screen "S2 Manual Mode" 1280x700, template "Navigation"
   on ClearScreen: SetBit("S2 Setup Data_Leave Manual Screen")
   on GenerateScreen: ResetBit("S2 Setup Data_Leave Manual Screen")
   Group "Group_3" at 492,12 size 427x42; Text 'SYSTEM 1'
   Group "Group_10" at 1149,100 size 112x111; Authorization "Health_Physics"
   Switch "Pushbutton_Emergency_1" at 935,29 size 60x61; CaptionText 'Switch'; TextOff '0'; TextOn '1'; PictureOff "Pushbutton_Emergency_Off_256c"; PictureOn "Pushbutton_Emergency_On_256c"
      Visibility <- "Station 2 Estop PB Active"
      ProcessValue <- "Station 2 Estop PB Active"
   TextField "Text field_53" at 933,7 size 65x25; Text 'ESTOP'
      Visibility <- "Station 2 Estop PB Active"
   Rectangle "Rectangle_4" at 411,100 size 720x467
      Appearance <- "Station 2 Run State"
   SymbolLibrary "Symbol library_18" at 680,195 size 148x16
      Appearance <- "Station 2 Tubing Rinse"
   SymbolLibrary "Symbol library_13" at 840,222 size 15x255
      Appearance <- "Station 2 Pump Tubing"
   SymbolLibrary "Symbol library_2" at 553,234 size 298x124
   SymbolLibrary "Symbol library_21" at 869,195 size 116x16
      Appearance <- "Station 2 Tubing Drain"
   TextField "Text field_9" at 590,186 size 85x32; Text 'RINSE'
   TextField "Text field_10" at 983,170 size 151x32; Text 'UNWANTED'
   TextField "Text field_14" at 828,471 size 38x32; Text 'SV'
   Group "Group_6" at 816,158 size 65x82
   Group "Group_12" at 916,230 size 108x188; TextOff 'WASTE'
   Group "Group_11" at 995,442 size 114x111; Authorization "Maintenance"
   TextField "Text field_17" at 984,192 size 135x32; Text 'MATERIAL'
   Group "Group" at 436,425 size 144x122
   Group "Group_4" at 629,370 size 156x40
   Group "Group_13" at 596,422 size 219x134; Text 'PUMP SPEED'; FormatPattern 99999
   Group "Group_14" at 1151,219 size 120x111; TextOff 'BYPASS'; Text 'DOOR LOCK'
   Group "Group_15" at 436,227 size 105x188
   Group "Group_9" at 482,274 size 532x42; Text 'SYSTEM 1'
   Group "Group_17" at 185,13 size 215x125; Authorization "Maintenance"
   IOField "I/O field_2" at 629,96 size 159x56; FormatPattern 9999.9
      ProcessValue <- "Station 2 MM Feedback RPM"
   TextField "Text field_8" at 629,64 size 165x32; Text 'PUMP SPEED'
   Rectangle "Rectangle_16" at 631,99 size 154x49
      Visibility <- "Station 2 Manual Mode"
   TextField "Text field_11" at 672,150 size 61x32; Text 'RPM'
   Group "Group_16" at 615,272 size 194x44
   Group "Group_18" at 615,272 size 194x44
   Group "Group_19" at 561,579 size 419x93
   Group "Group_20" at 561,579 size 419x93
   TextField "Text field_13" at 502,12 size 417x39; Text 'STATION 2 MANUAL MODE'
   Rectangle "Rectangle_11" at 482,274 size 518x42
      Visibility <- "Station 2 Process Running"
   TextField "Text field_16" at 494,274 size 520x39; Text 'STATION 2 IN AUTOMATIC MODE'
      Visibility <- "Station 2 Process Running"
   Rectangle "Rectangle_13" at 1149,100 size 112x111
      Visibility <- "CurrentGroupNum"
   TextField "Text field_15" at 1158,104 size 97x23; Text 'RAD LOCK'
      Visibility <- "CurrentGroupNum"
   Button "Button_15" at 1164,130 size 80x70; TextOff 'BYPASS'; Authorization "Health_Physics"
      on Press: InvertBit("Station 2 Rad Lock Bypass")
      Visibility <- "CurrentGroupNum"
   GraphicIOField "PlotLight_Round_GN_6" at 1218,132 size 22x23; PictureOn "PilotLight_Round_GN_On_256c"; PictureOff "PilotLight_Round_GN_Off_256c"; Authorization "Health_Physics"
      Visibility <- "CurrentGroupNum"
      ProcessValue <- "Station 2 Rad Lock Bypass"
   Group "Group_1" at 596,422 size 219x134; Text 'PUMP SPEED'; FormatPattern 99999
   Rectangle "Rectangle_12" at 629,463 size 154x49
      Visibility <- "Station 2 Manual Mode"
   IOField "I/O field_1" at 626,460 size 159x56; FormatPattern 9999.9
      ProcessValue <- "Station 2 Pump Speed RPM SP"
   TextField "Text field_5" at 607,428 size 205x32; Text 'PUMP SPEED SP'
   TextField "Text field_7" at 670,518 size 61x32; Text 'RPM'
   SymbolLibrary "Symbol library_4" at 816,185 size 32x36
      Appearance <- "Station 2 Valve Rinse"
   SymbolLibrary "Symbol library_3" at 849,185 size 32x36
      Appearance <- "Station 2 Valve Drain"
   SymbolLibrary "Symbol library_5" at 832,204 size 32x36
      Appearance <- "Station 2 Valve Pump"
   Group "Group_5" at 436,227 size 105x188
   Button "Button_9" at 449,264 size 74x63; TextOff 'FWD'
      Visibility <- "Station 2 Manual Mode"
   Button "Button_10" at 451,343 size 74x63; TextOff 'REV'
      Visibility <- "Station 2 Manual Mode"
   TextField "Text field_3" at 448,230 size 77x32; Text 'PUMP'
   Button "Button_5" at 449,264 size 74x63; TextOff 'FWD'
      on Press: SetBit("Station 2 MM Pump Dir FWD"); ResetBit("Station 2 MM Pump Dir REV")
   Button "Button_6" at 451,343 size 74x63; TextOff 'REV'
      on Press: SetBit("Station 2 MM Pump Dir REV"); ResetBit("Station 2 MM Pump Dir FWD")
   GraphicIOField "PlotLight_Round_GN_2" at 501,345 size 22x23; PictureOn "PilotLight_Round_GN_On_256c"; PictureOff "PilotLight_Round_GN_Off_256c"
      ProcessValue <- "Station 2 MM Pump Dir REV"
   GraphicIOField "PlotLight_Round_GN_5" at 500,266 size 22x23; PictureOn "PilotLight_Round_GN_On_256c"; PictureOff "PilotLight_Round_GN_Off_256c"
      ProcessValue <- "Station 2 MM Pump Dir FWD"
   Group "Group_2" at 916,230 size 108x188; TextOff 'WASTE'
   Button "Button_11" at 930,267 size 74x63; TextOff 'UM'
      Visibility <- "Station 2 Manual Mode"
   Button "Button_12" at 930,345 size 74x63; TextOff 'RINSE'
      Visibility <- "Station 2 Manual Mode"
   TextField "Text field_6" at 924,232 size 85x32; Text 'VALVE'
   Button "Button_7" at 930,267 size 74x63; TextOff 'UM'
      on Press: ResetBit("Station 2 MM Valve Direction SW")
   Button "Button_8" at 930,345 size 74x63; TextOff 'RINSE'
      on Press: SetBit("Station 2 MM Valve Direction SW")
   GraphicIOField "PlotLight_Round_GN_3" at 982,345 size 22x23; PictureOff "PilotLight_Round_GN_Off_256c"; PictureOn "PilotLight_Round_GN_On_256c"
      ProcessValue <- "Station 2 MM Valve Direction SW"
   GraphicIOField "PlotLight_Round_GN_4" at 980,267 size 22x23; PictureOn "PilotLight_Round_GN_Off_256c"; PictureOff "PilotLight_Round_GN_On_256c"
      ProcessValue <- "Station 2 MM Valve Direction SW"
   TextField "Text field_22" at 999,446 size 110x23; Text 'DOOR LOCK'
   Button "Button_16" at 1010,472 size 80x70; TextOff 'BYPASS'; Authorization "Maintenance"
      on Press: function_b14e0dd5("Station 2 Door Lock Open", 0)
   GraphicIOField "PlotLight_Round_GN_7" at 1064,474 size 22x23; PictureOn "PilotLight_Round_GN_On_256c"; PictureOff "PilotLight_Round_GN_Off_256c"; Authorization "Maintenance"
      ProcessValue <- "Station 2 Door Lock Open"
   TextField "Text field_18" at 440,429 size 140x32; Text 'PUMP RUN'
   Button "Button_17" at 471,463 size 74x63; TextOff 'SLEW'
      on Press: SetBit("Station 2 MM Pump Slew PB")
   GraphicIOField "PlotLight_Round_GN_8" at 520,465 size 22x23; PictureOff "PilotLight_Round_GN_Off_256c"; PictureOn "PilotLight_Round_GN_On_256c"
      ProcessValue <- "Station 2 MM Pump Slew PB"
   Group "Group_8" at 436,425 size 144x122; TextOff 'OFF'
   Button "Button_18" at 471,463 size 74x63; TextOff 'SLEW'
      Visibility <- "Station 2 Manual Mode"
   TextField "Text field_2" at 671,373 size 71x32; Text 'STOP'
      Visibility <- "Station 2 MM Pump Run"
   TextField "Text field_19" at 652,373 size 60x32; Text 'RUN'
      Visibility <- "Station 2 MM Pump Run"
   TextField "Text field_20" at 708,373 size 62x32; Text 'FWD'
      Visibility <- "Station 2 MM Pump FWD"
   TextField "Text field_21" at 711,373 size 55x32; Text 'REV'
      Visibility <- "Station 2 MM Pump REV"
   TextField "Text field_4" at 1152,223 size 119x21; Text 'RESET MOTOR'
   Button "Button_3" at 1168,249 size 80x70; TextOff 'RESET'
      on Press: InvertBit("Pump 2 Motor_Reset")
   GraphicIOField "PlotLight_Round_GN_9" at 1224,251 size 22x23; PictureOn "PilotLight_Round_GN_On_256c"; PictureOff "PilotLight_Round_GN_Off_256c"
      ProcessValue <- "Pump 2 Motor_Reset"
   TextField "Text field_1" at 201,18 size 194x32; Text 'MANUAL MODE'
   Button "Button_2" at 301,57 size 74x63; TextOff 'OFF'; Authorization "Maintenance"
      on Press: ResetBit("Station 2 Manual Mode"); SetTag("Station 2 Pump Speed RPM SP", 0); ResetBit("Station 2 MM Pump Dir FWD"); ResetBit("Station 2 MM Valve Direction SW"); ResetBit("Station 2 Warning 1"); ResetBit("Station 2 Warning 2"); ResetBit("Station 2 MM Pump Dir REV"); ResetBit("Station 2 Warning 1"); ResetBit("Station 2 Warning 2")
   Group "Group_7" at 207,57 size 74x63; Authorization "Maintenance"
   Button "Button_1" at 207,57 size 74x63; TextOff 'ON'; Authorization "Maintenance"
      on Press: SetBit("Station 2 Manual Mode")
      ObjectEnable <- "Station 2 Process Running"
   GraphicIOField "PlotLight_Round_GN" at 259,61 size 22x23; PictureOn "PilotLight_Round_GN_On_256c"; PictureOff "PilotLight_Round_GN_Off_256c"; Authorization "Maintenance"
      ProcessValue <- "Station 2 Manual Mode"
   Rectangle "Rectangle_17" at 615,274 size 194x42
      Visibility <- "Station 2 Warning 1"
   TextField "Text field_27" at 630,272 size 164x43; Text 'CAUTION'
      Visibility <- "Station 2 Warning 1"
   Rectangle "Rectangle_8" at 615,274 size 194x42
      Visibility <- "Station 2 Warning 2"
   TextField "Text field_12" at 630,272 size 164x43; Text 'CAUTION'
      Visibility <- "Station 2 Warning 2"
   TextField "Text field_28" at 588,579 size 354x37; Text 'Material will be pumped'
      Visibility <- "Station 2 Warning 2"
   TextField "Text field_29" at 630,607 size 257x37; Text 'from SV to Rinse.'
      Visibility <- "Station 2 Warning 2"
   TextField "Text field_30" at 561,635 size 419x37; Text 'Material may be radioactive!'
      Visibility <- "Station 2 Warning 2"
   TextField "Text field_23" at 588,579 size 354x37; Text 'Material will be pumped'
      Visibility <- "Station 2 Warning 1"
   TextField "Text field_24" at 619,607 size 279x37; Text 'from UM to the SV.'
      Visibility <- "Station 2 Warning 1"
   TextField "Text field_25" at 561,635 size 419x37; Text 'Material may be radioactive!'
      Visibility <- "Station 2 Warning 1"

screen "User Control" 1280x700, template "Navigation"
   UserView "User view_1" at 220,70 size 927x482
   Button "SB_ExitRuntime_53x53" at 1198,17 size 53x53; TextOff 'Text'; Authorization "User administration"; PictureOff "SB_ExitRuntime_53x53_256c"
      on Click: StopRuntime(0)
   Group "Group_3" at 542,17 size 257x42; Text 'SYSTEM 1'
   TextField "Text field_13" at 548,17 size 245x39; Text 'USER CONTROL'

screen "Rad Settings" 1280x700, template "Navigation"
   Group "Group_1" at 505,20 size 445x49; Text 'SYSTEM 1'
   Group "Group_6" at 299,526 size 301x91; FormatPattern 9999.9
   TextField "Text field_29" at 343,99 size 221x29; Text 'ALARM SETPOINTS'
   Group "Group_3" at 746,131 size 320x136; Picture "Graphic_1"; FormatPattern 9999.9
   Group "Group_8" at 748,327 size 320x137; Picture "Graphic_1"; FormatPattern 9999.9
   Group "Group" at 749,526 size 320x76; Picture "Graphic_1"; FormatPattern 9999.9
   TextField "Text field_4" at 787,99 size 242x29; Text 'CURRENT READINGS'
   Group "Group_5" at 297,131 size 301x186; FormatPattern 9999.9
   Group "Group_2" at 298,327 size 301x186; FormatPattern 9999.9
   TextField "Text field_15" at 512,20 size 438x43; Text 'RAD SETTINGS (uRem/h)'
   TextField "Text field_12" at 376,139 size 128x29; Text 'STATION 1'
   TextField "Text field_17" at 302,195 size 157x27; Text 'ALARM LEVEL:'
   IOField "I/O field_8" at 452,241 size 137x48; FormatPattern 999999
      ProcessValue <- "Station 1 Pump Rad Alarm Level"
   TextField "Text field_18" at 304,239 size 64x27; Text 'PUMP'
   IOField "I/O field_1" at 450,174 size 139x48; FormatPattern 999999
      ProcessValue <- "Station 1 Vessel Rad Alarm Level"
   TextField "Text field_1" at 302,259 size 157x27; Text 'ALARM LEVEL:'
   TextField "Text field_2" at 302,174 size 83x27; Text 'VESSEL'
   IOField "I/O field_3" at 452,549 size 136x48; FormatPattern 999999
      ProcessValue <- "Waste Rad High Alarm"
   Group "Group_4" at 307,536 size 157x67
   TextField "Text field_6" at 308,536 size 128x27; Text 'UNWANTED'
   TextField "Text field_26" at 308,556 size 114x27; Text 'MATERIAL'
   TextField "Text field_5" at 307,576 size 157x27; Text 'ALARM LEVEL:'
   TextField "Text field_9" at 380,334 size 128x29; Text 'STATION 2'
   IOField "I/O field_5" at 450,439 size 135x48; FormatPattern 999999
      ProcessValue <- "Station 2 Pump Rad Alarm Level"
   IOField "I/O field_10" at 450,371 size 135x48; FormatPattern 999999
      ProcessValue <- "Station 2 Vessel Rad Alarm Level"
   TextField "Text field_16" at 303,455 size 157x27; Text 'ALARM LEVEL:'
   TextField "Text field_21" at 304,372 size 83x27; Text 'VESSEL'
   TextField "Text field_11" at 304,434 size 64x27; Text 'PUMP'
   TextField "Text field_10" at 304,392 size 157x27; Text 'ALARM LEVEL:'
   TextField "Text field_3" at 758,171 size 128x25; Text 'VESSEL CAVE'
   TextField "Text field_46" at 773,215 size 113x25; Text 'PUMP CAVE'
   TextField "Text field_49" at 808,134 size 120x27; Text 'STATION 1'
   TextField "Text field_50" at 923,133 size 109x27; Text '(uRem/h)'
   IOField "I/O field_13" at 888,166 size 113x34; FormatPattern 999999
      ProcessValue <- "Station 1 Vessel Rad Level"
   IOField "I/O field_15" at 888,210 size 113x34; FormatPattern 999999
      ProcessValue <- "Station 1 Pump Rad Level"
   GraphicView "Graphic view_2" at 1009,164 size 36x36; Picture "Graphic_1"
      Visibility <- "Station 1 Vessel Rad Alarm"
   GraphicView "Graphic view_1" at 1009,208 size 36x36; Picture "Graphic_1"
      Visibility <- "Station 1 Pump Rad Alarm"
   TextField "Text field_51" at 764,365 size 128x25; Text 'VESSEL CAVE'
   TextField "Text field_54" at 775,409 size 113x25; Text 'PUMP CAVE'
   TextField "Text field_57" at 808,330 size 120x27; Text 'STATION 2'
   TextField "Text field_58" at 923,329 size 109x27; Text '(uRem/h)'
   IOField "I/O field_16" at 888,361 size 112x34; FormatPattern 999999
      ProcessValue <- "Station 2 Vessel Rad Level"
   IOField "I/O field_17" at 888,406 size 112x34; FormatPattern 999999
      ProcessValue <- "Station 2 Pump Rad Level"
   GraphicView "Graphic view_6" at 1008,359 size 36x36; Picture "Graphic_1"
      Visibility <- "Station 2 Vessel Rad Alarm"
   GraphicView "Graphic view_4" at 1009,405 size 36x36; Picture "Graphic_1"
      Visibility <- "Station 2 Pump Rad Alarm"
   TextField "Text field_47" at 775,534 size 114x25; Text 'UNWANTED'
   IOField "I/O field_18" at 894,556 size 112x34; FormatPattern 999999
      ProcessValue <- "Waste Rad Level"
   GraphicView "Graphic view_3" at 1012,544 size 36x36; Picture "Graphic_1"
      Visibility <- "Waste Rad Alarm"
   TextField "Text field_19" at 785,552 size 102x25; Text 'MATERIAL'
   TextField "Text field_20" at 815,570 size 66x25; Text 'VAULT'
   TextField "Text field_33" at 900,531 size 93x23; Text '(uRem/h)'

screen "Alarm Screen" 1280x700, template "Navigation"
   AlarmView "Alarm view_1" at 210,51 size 1021x325
   Group "Group_3" at 552,3 size 222x42; Text 'SYSTEM 1'
   AlarmView "Alarm view_2" at 211,416 size 1020x262
   TextField "Text field_1" at 239,386 size 210x34; Text 'ALARM BUFFER'
   TextField "Text field_13" at 557,3 size 210x39; Text 'ALARM VIEW'

screen "Status" 1280x700, template "Navigation"
   Group "Group_4" at 223,19 size 217x247
   Group "Group_3" at 1012,378 size 245x42; Text 'SYSTEM 1'
   Group "Group_2" at 1023,427 size 226x122; PictureOff "PilotLight_Round_G_Off_256c"; PictureOn "PilotLight_Round_R_On_256c"
   Group "Group_6" at 1023,555 size 226x122; PictureOff "PilotLight_Round_G_Off_256c"; PictureOn "PilotLight_Round_R_On_256c"
   Group "Group_8" at 192,279 size 261x74
   Group "Group_5" at 463,11 size 545x342
   Group "Group_9" at 1000,11 size 273x342
   Rectangle "Rectangle_9" at 1001,11 size 273x684
      Visibility <- "CurrentGroupNum"
   Group "Group_28" at 527,378 size 117x42; Text 'SYSTEM 1'
   Group "Group_1" at 251,432 size 320x136; Picture "Graphic_1"; FormatPattern 9999.9
   Group "Group" at 434,586 size 320x76; Picture "Graphic_1"; FormatPattern 9999.9
   Group "Group_7" at 596,432 size 320x137; Picture "Graphic_1"; FormatPattern 9999.9
   Button "Template_Button_3" at 246,85 size 166x69; TextOff 'S1 SETTINGS'
      on Press: function_efd93a16("Station 1 Settings", 180, 100, -1, -1, 1)
   Button "Template_Button_1" at 246,175 size 166x69; TextOff 'S2 SETTINGS'
      on Press: function_efd93a16("Station 2 Settings", 180, 100, -1, -1, 1)
   TextField "Text field_1" at 230,25 size 210x27; Text 'CURRENT PROCESS'
   TextField "Text field_2" at 270,45 size 111x27; Text 'SETTINGS'
   IOField "I/O field_1" at 707,96 size 128x48; FormatPattern 999.99
      ProcessValue <- "Station 1 Total Water Supply Volume"
   TextField "Text field_3" at 474,108 size 183x29; Text 'WATER SUPPLY'
   TextField "Text field_6" at 837,107 size 18x29; Text 'L'
   TextField "Text field_8" at 474,86 size 244x29; Text 'STATION 1 CURRENT'
   Button "Button_1" at 874,76 size 98x74; TextOff 'S1 H20 RESET'
      on Press: function_efd93a16("S1 Container Change", 680, 360, -1, -1, 1)
      ObjectEnable <- "Station 1 Process Running"
   IOField "I/O field_2" at 709,189 size 128x48; FormatPattern 999.99
      ProcessValue <- "Station 2 Total Water Supply Volume"
   TextField "Text field_4" at 476,201 size 183x29; Text 'WATER SUPPLY'
   TextField "Text field_5" at 476,179 size 244x29; Text 'STATION 2 CURRENT'
   Button "Button_2" at 876,169 size 98x74; TextOff 'S2 H20 RESET'
      on Press: function_efd93a16("S2 Container Change", 680, 360, -1, -1, 1)
      ObjectEnable <- "Station 2 Process Running"
   TextField "Text field_7" at 838,200 size 18x29; Text 'L'
   IOField "I/O field_3" at 708,281 size 128x48; FormatPattern 999.99
      ProcessValue <- "Total Waste Drum Volume"
   TextField "Text field_9" at 475,297 size 197x29; Text 'SUPPLY VOLUME'
   TextField "Text field_10" at 475,276 size 235x29; Text 'UM DRUM CURRENT'
   Button "Button_3" at 875,261 size 98x74; TextOff 'UM RESET'
      on Press: function_efd93a16("UM Container Change", 680, 360, -1, -1, 1)
   TextField "Text field_11" at 837,292 size 18x29; Text 'L'
   TextField "Text field_12" at 826,20 size 182x27; Text 'FOR CONTAINER'
   TextField "Text field_13" at 832,42 size 158x27; Text 'CHANGE ONLY'
   TextField "Text field_25" at 474,130 size 101x29; Text 'VOLUME'
   TextField "Text field_26" at 476,222 size 101x29; Text 'VOLUME'
   GraphicIOField "PlotLight_Round_R" at 1183,459 size 33x31; PictureOff "PilotLight_Round_G_Off_256c"; PictureOn "PilotLight_Round_R_On_256c"
      ProcessValue <- "Station 1 Pump Error Code Bit"
   TextField "Text field_16" at 1031,461 size 148x25; Text 'ERROR STATUS'
   TextField "Text field_17" at 1032,503 size 126x25; Text 'ERROR CODE'
   TextField "Text field_18" at 1085,430 size 120x27; Text 'STATION 1'
   IOField "I/O field_5" at 1170,499 size 60x34; FormatPattern 999
      ProcessValue <- "Station 1 Pump Error Code"
   TextField "Text field_22" at 1026,378 size 223x39; Text 'PUMP STATUS'
   GraphicIOField "PlotLight_Round_R_1" at 1183,587 size 33x31; PictureOn "PilotLight_Round_R_On_256c"; PictureOff "PilotLight_Round_G_Off_256c"
      ProcessValue <- "Station 2 Pump Error Code Bit"
   TextField "Text field_21" at 1031,589 size 148x25; Text 'ERROR STATUS'
   TextField "Text field_23" at 1032,631 size 126x25; Text 'ERROR CODE'
   TextField "Text field_24" at 1085,558 size 120x27; Text 'STATION 2'
   IOField "I/O field_4" at 1170,627 size 60x34; FormatPattern 999
      ProcessValue <- "Station 2 Pump Error Code"
   TextField "Text field_27" at 231,282 size 193x27; Text 'SYSTEM VERSION'
   IOField "I/O field_8" at 198,311 size 246x28; FormatPattern ????????????????????
      ProcessValue <- "System Version"
   IOField "I/O field_9" at 1011,96 size 128x48; FormatPattern 999.99
      ProcessValue <- "Station 1 Total Water Supply Update"
   TextField "Text field_28" at 1049,20 size 200x27; Text 'CORRECT VOLUME'
   TextField "Text field_29" at 1076,42 size 141x27; Text 'MAINT ONLY'
   TextField "Text field_30" at 1140,108 size 18x29; Text 'L'
   Button "Button_4" at 1164,75 size 98x74; TextOff 'S1 H20 UPDATE'
      on Press: SetBit("Station 1 Water Update")
      ObjectEnable <- "Station 1 Process Running"
   IOField "I/O field_10" at 1012,187 size 128x48; FormatPattern 999.99
      ProcessValue <- "Station 2 Total Water Supply Update"
   Button "Button_5" at 1164,169 size 98x74; TextOff 'S2 H20 UPDATE'
      on Press: SetBit("Station 2 Water Update")
      ObjectEnable <- "Station 2 Process Running"
   TextField "Text field_31" at 1139,201 size 18x29; Text 'L'
   IOField "I/O field_11" at 1012,279 size 128x48; FormatPattern 999.99
      ProcessValue <- "Total Waste Drum Update"
   TextField "Text field_32" at 1143,290 size 18x29; Text 'L'
   Button "Button_6" at 1164,261 size 98x74; TextOff 'UM UPDATE'
      on Press: SetBit("Waste Drum Update")
   TextField "Text field_14" at 539,378 size 94x39; Text 'ALMO'
   TextField "Text field_15" at 263,472 size 128x25; Text 'VESSEL CAVE'
   TextField "Text field_46" at 278,516 size 113x25; Text 'PUMP CAVE'
   TextField "Text field_49" at 313,435 size 120x27; Text 'STATION 1'
   TextField "Text field_50" at 428,434 size 109x27; Text '(uRem/h)'
   IOField "I/O field_13" at 393,467 size 113x34; FormatPattern 999999
      ProcessValue <- "Station 1 Vessel Rad Level"
   IOField "I/O field_15" at 393,511 size 113x34; FormatPattern 999999
      ProcessValue <- "Station 1 Pump Rad Level"
   GraphicView "Graphic view_2" at 514,465 size 36x36; Picture "Graphic_1"
      Visibility <- "Station 1 Vessel Rad Alarm"
   GraphicView "Graphic view_1" at 514,509 size 36x36; Picture "Graphic_1"
      Visibility <- "Station 1 Pump Rad Alarm"
   TextField "Text field_51" at 612,470 size 128x25; Text 'VESSEL CAVE'
   TextField "Text field_54" at 623,514 size 113x25; Text 'PUMP CAVE'
   TextField "Text field_57" at 656,435 size 120x27; Text 'STATION 2'
   TextField "Text field_58" at 771,434 size 109x27; Text '(uRem/h)'
   IOField "I/O field_16" at 736,466 size 112x34; FormatPattern 999999
      ProcessValue <- "Station 2 Vessel Rad Level"
   IOField "I/O field_17" at 736,511 size 112x34; FormatPattern 999999
      ProcessValue <- "Station 2 Pump Rad Level"
   GraphicView "Graphic view_6" at 856,464 size 36x36; Picture "Graphic_1"
      Visibility <- "Station 2 Vessel Rad Alarm"
   GraphicView "Graphic view_4" at 857,510 size 36x36; Picture "Graphic_1"
      Visibility <- "Station 2 Pump Rad Alarm"
   TextField "Text field_47" at 460,594 size 114x25; Text 'UNWANTED'
   IOField "I/O field_18" at 579,616 size 112x34; FormatPattern 999999
      ProcessValue <- "Waste Rad Level"
   GraphicView "Graphic view_3" at 697,604 size 36x36; Picture "Graphic_1"
      Visibility <- "Waste Rad Alarm"
   TextField "Text field_19" at 470,612 size 102x25; Text 'MATERIAL'
   TextField "Text field_20" at 500,630 size 66x25; Text 'VAULT'
   TextField "Text field_33" at 585,591 size 93x23; Text '(uRem/h)'

Template "Navigation" 1280x700
   Button "Template_Button_3" at 35,8 size 130x55; TextOff 'HOME'
      on Press: ActivateScreen("Home Screen", 0)
   Button "Template_Button_5" at 35,143 size 130x55; TextOff 'STATUS'
      on Press: ActivateScreen("Status", 0)
   Button "Template_Button_9" at 36,563 size 130x55; TextOff 'USER CONTROL'
      on Press: ActivateScreen("User Control", 0)
      Visibility <- "CurrentGroupNum"
   Button "Template_Button_4" at 35,75 size 130x55; TextOff 'ALARMS'
      on Press: ActivateScreen("Alarm Screen", 0)
   Rectangle "Template_Rectangle_1" at 27,209 size 147x272
      Visibility <- "CurrentGroupNum"
   Button "Template_Button_1" at 35,215 size 130x55; TextOff 'STATION 1 MANUAL'; Authorization "Maintenance"
      on Click: ActivateScreen("S1 Manual Mode", 0)
      Visibility <- "CurrentGroupNum"
   Button "Template_Button_2" at 35,351 size 130x55; TextOff 'STATION 1 SETUP'; Authorization "Maintenance"
      on Press: ActivateScreen("S1 Setup Screen", 0)
      Visibility <- "CurrentGroupNum"
   Button "Template_Button_7" at 35,419 size 130x55; TextOff 'STATION 2 SETUP'; Authorization "Maintenance"
      on Press: ActivateScreen("S2 Setup Screen", 0)
      Visibility <- "CurrentGroupNum"
   Button "Template_Button_8" at 35,283 size 130x55; TextOff 'STATION 2 MANUAL'; Authorization "Maintenance"
      on Press: ActivateScreen("S2 Manual Mode", 0)
      Visibility <- "CurrentGroupNum"
   Button "Template_Button_6" at 35,494 size 130x55; TextOff 'RAD SETTINGS'; Authorization "Maintenance"
      on Press: ActivateScreen("Rad Settings", 0)
      Visibility <- "CurrentGroupNum"

PopupScreen "Station 1 Settings" 1050x700
   TextField "Text field_15" at 199,16 size 372x43; Text 'STATION 1 SETTINGS'
   Button "Template_Button_3" at 37,480 size 166x69; TextOff 'RETURN'
      on Press: function_efd93a16()
   Group "Group_5" at 190,16 size 385x49; Text 'SYSTEM 1'
   Group "Group" at 34,91 size 275x295; Authorization "Maintenance"
   Group "Group_2" at 348,91 size 275x235; Authorization "Maintenance"
   Group "Group_7" at 661,32 size 275x164; Authorization "Maintenance"
   Group "Group_3" at 661,195 size 275x164; Authorization "Maintenance"
   Group "Group_4" at 661,358 size 275x164; Authorization "Maintenance"
   TextField "Text field_12" at 65,96 size 206x29; Text 'PROCESS TIMERS'
   TextField "Text field_16" at 39,314 size 129x27; Text 'TOTAL NUM'
   IOField "I/O field_7" at 162,319 size 130x48; Authorization "Maintenance"; FormatPattern 999
      ProcessValue <- "S1 Auto Number of Rinses"
   TextField "Text field_17" at 39,275 size 124x27; Text 'TIME (ms):'
   IOField "I/O field_8" at 161,256 size 130x48; Authorization "Maintenance"; FormatPattern 99999
      ProcessValue <- "S1 Auto Rinse Run Time"
   TextField "Text field_18" at 38,253 size 72x27; Text 'RINSE'
   IOField "I/O field_9" at 160,194 size 130x48; Authorization "Maintenance"; FormatPattern 99999
      ProcessValue <- "S1 Auto Drain Run Time"
   TextField "Text field_19" at 39,191 size 75x27; Text 'DRAIN'
   TextField "Text field_20" at 40,213 size 124x27; Text 'TIME (ms):'
   TextField "Text field_21" at 39,337 size 93x27; Text 'CYCLES:'
   IOField "I/O field_18" at 160,133 size 130x48; Authorization "Maintenance"; FormatPattern 99999
      ProcessValue <- "S1 Auto Remove Run Time"
   TextField "Text field_41" at 39,130 size 94x27; Text 'REMOVE'
   TextField "Text field_42" at 40,152 size 124x27; Text 'TIME (ms):'
   TextField "Text field_4" at 381,95 size 210x29; Text 'PUMP MAX SPEED'
   TextField "Text field_5" at 377,204 size 83x27; Text 'DRAIN:'
   IOField "I/O field_1" at 455,196 size 101x48; Authorization "Maintenance"; FormatPattern 999
      ProcessValue <- "S1 Auto Pump Drain Max Speed"
   TextField "Text field_6" at 378,269 size 80x27; Text 'RINSE:'
   IOField "I/O field_2" at 455,260 size 101x48; Authorization "Maintenance"; FormatPattern 999
      ProcessValue <- "S1 Auto Pump Rinse Max Speed"
   TextField "Text field_13" at 554,269 size 51x27; Text 'RPM'
   TextField "Text field_14" at 555,204 size 51x27; Text 'RPM'
   TextField "Text field_37" at 360,141 size 102x27; Text 'REMOVE:'
   IOField "I/O field_17" at 454,133 size 101x48; Authorization "Maintenance"; FormatPattern 999
      ProcessValue <- "S1 Auto Pump Remove Max Speed"
   TextField "Text field_38" at 554,141 size 51x27; Text 'RPM'
   TextField "Text field_43" at 713,36 size 174x29; Text 'REMOVE RAMP'
   TextField "Text field_49" at 675,80 size 124x27; Text 'NO. STEPS:'
   IOField "I/O field_19" at 792,72 size 128x48; Authorization "Maintenance"; FormatPattern 999
      ProcessValue <- "S1Auto Ramp Remove Step"
   TextField "Text field_50" at 674,141 size 124x27; Text 'TIME (ms):'
   IOField "I/O field_22" at 791,134 size 128x48; Authorization "Maintenance"; FormatPattern 99999
      ProcessValue <- "S1Auto Ramp Remove Time"
   TextField "Text field_1" at 724,199 size 154x29; Text 'DRAIN RAMP'
   TextField "Text field_7" at 674,243 size 124x27; Text 'NO. STEPS:'
   IOField "I/O field_3" at 791,235 size 128x48; Authorization "Maintenance"; FormatPattern 999
      ProcessValue <- "S1 Auto Ramp Drain Step"
   TextField "Text field_8" at 673,304 size 124x27; Text 'TIME (ms):'
   IOField "I/O field_4" at 790,297 size 128x48; Authorization "Maintenance"; FormatPattern 99999
      ProcessValue <- "S1 Auto Ramp Drain Time"
   TextField "Text field_9" at 728,362 size 150x29; Text 'RINSE RAMP'
   TextField "Text field_10" at 672,408 size 124x27; Text 'NO. STEPS:'
   IOField "I/O field_5" at 792,398 size 125x48; Authorization "Maintenance"; FormatPattern 999
      ProcessValue <- "S1 Auto Ramp Rinse Step"
   TextField "Text field_11" at 671,467 size 124x27; Text 'TIME (ms):'
   IOField "I/O field_6" at 793,460 size 125x48; Authorization "Maintenance"; FormatPattern 99999
      ProcessValue <- "S1 Auto Ramp Rinse Time"

PopupScreen "Station 2 Settings" 1050x700
   TextField "Text field_15" at 225,19 size 372x43; Text 'STATION 2 SETTINGS'
   Button "Template_Button_3" at 50,453 size 166x69; TextOff 'RETURN'
      on Press: function_efd93a16()
   Group "Group_1" at 216,19 size 381x49; Text 'SYSTEM 1'
   Group "Group_3" at 672,182 size 264x164; Text 'WASTE RAMP'; Authorization "Maintenance"
   Group "Group_4" at 672,345 size 265x164; Authorization "Maintenance"
   Group "Group" at 56,76 size 275x290; Authorization "Maintenance"
   Group "Group_2" at 370,76 size 275x227; Authorization "Maintenance"
   Group "Group_7" at 672,19 size 264x164; Authorization "Maintenance"
   TextField "Text field_1" at 737,186 size 154x29; Text 'DRAIN RAMP'
   TextField "Text field_7" at 677,230 size 124x27; Text 'NO. STEPS:'
   IOField "I/O field_3" at 794,222 size 128x48; Authorization "Maintenance"; FormatPattern 999
      ProcessValue <- "S2 Auto Ramp Drain Step"
   TextField "Text field_8" at 676,291 size 124x27; Text 'TIME (ms):'
   IOField "I/O field_4" at 793,284 size 128x48; Authorization "Maintenance"; FormatPattern 99999
      ProcessValue <- "S2 Auto Ramp Drain Time"
   TextField "Text field_9" at 739,349 size 150x29; Text 'RINSE RAMP'
   TextField "Text field_10" at 678,395 size 124x27; Text 'NO. STEPS:'
   IOField "I/O field_5" at 798,385 size 125x48; Authorization "Maintenance"; FormatPattern 999
      ProcessValue <- "S2 Auto Ramp Rinse Step"
   TextField "Text field_11" at 677,454 size 124x27; Text 'TIME (ms):'
   IOField "I/O field_6" at 799,447 size 125x48; Authorization "Maintenance"; FormatPattern 99999
      ProcessValue <- "S2 Auto Ramp Rinse Time"
   TextField "Text field_12" at 95,81 size 206x29; Text 'PROCESS TIMERS'
   TextField "Text field_16" at 61,299 size 129x27; Text 'TOTAL NUM'
   IOField "I/O field_7" at 184,304 size 130x48; Authorization "Maintenance"; FormatPattern 999
      ProcessValue <- "S2 Auto Number of Rinses"
   TextField "Text field_17" at 61,260 size 124x27; Text 'TIME (ms):'
   IOField "I/O field_8" at 183,241 size 130x48; Authorization "Maintenance"; FormatPattern 99999
      ProcessValue <- "S2 Auto Rinse Run Time"
   TextField "Text field_18" at 60,238 size 72x27; Text 'RINSE'
   IOField "I/O field_9" at 182,179 size 130x48; Authorization "Maintenance"; FormatPattern 99999
      ProcessValue <- "S2 Auto Drain Run Time"
   TextField "Text field_19" at 61,176 size 75x27; Text 'DRAIN'
   TextField "Text field_20" at 62,198 size 124x27; Text 'TIME (ms):'
   TextField "Text field_21" at 61,322 size 93x27; Text 'CYCLES:'
   IOField "I/O field_15" at 182,117 size 130x48; Authorization "Maintenance"; FormatPattern 99999
      ProcessValue <- "S2 Auto Remove Run Time"
   TextField "Text field_34" at 61,114 size 94x27; Text 'REMOVE'
   TextField "Text field_35" at 62,136 size 124x27; Text 'TIME (ms):'
   TextField "Text field_4" at 407,80 size 210x29; Text 'PUMP MAX SPEED'
   TextField "Text field_5" at 393,182 size 83x27; Text 'DRAIN:'
   IOField "I/O field_1" at 476,174 size 101x48; Authorization "Maintenance"; FormatPattern 999
      ProcessValue <- "S2 Auto Pump Drain Max Speed"
   TextField "Text field_6" at 398,243 size 80x27; Text 'RINSE:'
   IOField "I/O field_2" at 477,236 size 101x48; Authorization "Maintenance"; FormatPattern 999
      ProcessValue <- "S2 Auto Pump Rinse Max Speed"
   TextField "Text field_13" at 581,243 size 51x27; Text 'RPM'
   TextField "Text field_14" at 579,182 size 51x27; Text 'RPM'
   TextField "Text field_36" at 376,120 size 102x27; Text 'REMOVE:'
   IOField "I/O field_17" at 476,112 size 101x48; Authorization "Maintenance"; FormatPattern 999
      ProcessValue <- "S2 Auto Pump Remove Max Speed"
   TextField "Text field_37" at 579,120 size 51x27; Text 'RPM'
   TextField "Text field_38" at 726,23 size 174x29; Text 'REMOVE RAMP'
   TextField "Text field_41" at 677,67 size 124x27; Text 'NO. STEPS:'
   IOField "I/O field_18" at 794,59 size 128x48; Authorization "Maintenance"; FormatPattern 999
      ProcessValue <- "S2 Auto Ramp Remove Step"
   TextField "Text field_42" at 676,128 size 124x27; Text 'TIME (ms):'
   IOField "I/O field_19" at 793,121 size 128x48; Authorization "Maintenance"; FormatPattern 99999
      ProcessValue <- "S2 Auto Ramp Remove Time"

PopupScreen "S1 Container Change" 400x400
   Button "Template_Button_3" at 145,301 size 166x69; TextOff 'RETURN'
      on Press: function_efd93a16()
   TextField "Text field_1" at 31,42 size 330x29; Text 'Have you changed the water'
   TextField "Text field_2" at 36,65 size 318x29; Text 'container and wish to reset'
   TextField "Text field_3" at 82,159 size 86x47; Text 'YES:'
   Button "Button_1" at 178,145 size 98x74; TextOff 'RESET'
      on Press: SetBit("Station 1 New Water Container"); ActivateScreen("Status", 0)
      ObjectEnable <- "Station 1 Run State"
   TextField "Text field_4" at 70,314 size 70x43; Text 'NO:'
   TextField "Text field_5" at 27,88 size 349x29; Text 'the current container volume?'
   TextField "Text field_6" at 136,10 size 128x29; Text 'STATION 1'

PopupScreen "S2 Container Change" 400x400
   Button "Template_Button_3" at 145,301 size 166x69; TextOff 'RETURN'
      on Press: function_efd93a16()
   TextField "Text field_1" at 44,42 size 330x29; Text 'Have you changed the water'
   TextField "Text field_2" at 52,65 size 318x29; Text 'container and wish to reset'
   TextField "Text field_3" at 82,159 size 86x47; Text 'YES:'
   Button "Button_1" at 178,145 size 98x74; TextOff 'RESET'
      on Press: SetBit("Station 2 New Water Container"); ActivateScreen("Status", 0)
      ObjectEnable <- "Station 2 Run State"
   TextField "Text field_4" at 70,314 size 70x43; Text 'NO:'
   TextField "Text field_5" at 42,88 size 349x29; Text 'the current container volume?'
   TextField "Text field_6" at 136,10 size 128x29; Text 'STATION 2'

PopupScreen "UM Container Change" 400x400
   Button "Template_Button_3" at 145,301 size 166x69; TextOff 'RETURN'
      on Press: function_efd93a16()
   TextField "Text field_1" at 62,42 size 300x29; Text 'Have you changed the UM'
   TextField "Text field_2" at 57,65 size 318x29; Text 'container and wish to reset'
   TextField "Text field_3" at 82,159 size 86x47; Text 'YES:'
   Button "Button_1" at 178,145 size 98x74; TextOff 'RESET'
      on Press: SetBit("Station 1 New Waste Container"); SetBit("Station 2 New Waste Container"); ActivateScreen("Status", 0)
      ObjectEnable <- "Station 1 Run State"
   TextField "Text field_4" at 70,314 size 70x43; Text 'NO:'
   TextField "Text field_5" at 47,88 size 349x29; Text 'the current container volume?'
   TextField "Text field_6" at 80,10 size 264x29; Text 'UNWANTED MATERIAL'

screen "Future" 1280x700
   Group "Group_13" at 435,105 size 80x70; TextOff 'RAD CTRL'; Authorization "Maintenance"
   TextField "Text field_33" at 432,71 size 283x29; Text 'CONTROL TO RAD LEVEL'
   IOField "I/O field_20" at 552,126 size 130x48; Authorization "Maintenance"; FormatPattern 9999.9
      ProcessValue <- "S2 Auto Rinse to RAD Level"
   TextField "Text field_34" at 534,100 size 195x22; Text 'RAD LEVEL SP (uSv/h)'
   Button "Button_1" at 435,105 size 80x70; TextOff 'AUTO RAD CTRL'; Authorization "Maintenance"
      on Press: InvertBit("S2 Auto Use RAD CTRL")
   GraphicIOField "PlotLight_Round_GN_1" at 489,107 size 22x23; PictureOn "PilotLight_Round_GN_On_256c"; PictureOff "PilotLight_Round_GN_Off_256c"; Authorization "Maintenance"
      ProcessValue <- "S2 Auto Use RAD CTRL"
   Group "Group_14" at 414,71 size 315x121; TextOff 'RAD CTRL'; Text 'RINSE TO RAD LEVEL'; Authorization "Maintenance"; FormatPattern 9999
   Group "Group_12" at 414,209 size 315x121; TextOff 'RAD CTRL'; Text 'RINSE TO RAD LEVEL'; Authorization "Maintenance"; FormatPattern 9999
   Group "Group_11" at 435,243 size 80x70; TextOff 'RAD CTRL'; Authorization "Maintenance"
   TextField "Text field_39" at 430,209 size 283x29; Text 'CONTROL TO RAD LEVEL'
   IOField "I/O field_19" at 552,264 size 130x48; Authorization "Maintenance"; FormatPattern 9999.9
      ProcessValue <- "S1 Auto Rinse to RAD Level"
   TextField "Text field_40" at 534,238 size 195x22; Text 'RAD LEVEL SP (uSv/h)'
   Button "Button_15" at 435,243 size 80x70; TextOff 'AUTO RAD CTRL'; Authorization "Maintenance"
      on Press: InvertBit("S1 Auto Use RAD CTRL")
   GraphicIOField "PlotLight_Round_GN_6" at 489,245 size 22x23; PictureOn "PilotLight_Round_GN_On_256c"; PictureOff "PilotLight_Round_GN_Off_256c"; Authorization "Maintenance"
      ProcessValue <- "S1 Auto Use RAD CTRL"

VB script "TitleUpdater"
   Dim title
   Set title = HmiRuntime.Screens(0).ScreenItems("Screen title")
   title.Text = HmiRuntime.BaseScreenName

scheduled task "Get User Name"
   on Action: function_f41c6f6c("CurrentUserName"); function_e1ab61de("CurrentGroupNum")
*)